INTERFACE I_Display

METHOD PUBLIC UpdateFrom
VAR_INPUT
	Source : I_ReadableDisplayBuffer;
END_VAR
END_METHOD

END_INTERFACE

(* stored: Version 1.1.0.1, ProductVersion 3.1.4024.15
   Itf I_Display: Id {89d9bb48-c0f1-47f0-9295-3b71725380eb}
   Method UpdateFrom: Id {5e5c81c5-3c57-4c66-b04b-e338a6f3e647} *)
